FUNCTION_BLOCK Q_GraphicsContext (* Command Graphics Context ( Part 6 - F.56 ) *)
  (* Standard: ISO 11783-6; Description: Copyright (c) 2022 HR Agrartechnik GmbH This program and the accompanying materials are made available under the terms of the Eclipse Public License 2.0 which is available at https://www.eclipse.org/legal/epl-2.0/ SPDX-License-Identifier: EPL-2.0 see Description Tab *)
  (* Version 1.0, 2022-07-08, Franz Höpfinger, HR Agrartechnik GmbH *)
  PACKAGE isobus::UT::Q;
  IMPORT eclipse4diac::core::TypeHash;
  IMPORT isobus::UT::Q::IDs::ID_NULL;
  (* Documentation:
  Command Graphics Context ( Part 6 - F.56 )
   This command is used to manipulate a graphics Context object (only on version 4 or later VTs).
   param[in] {objectID, uint16_t}
   Object ID of a Graphics Context object
   param[in] {SubCommandID, uint8_t}
   Sub-Command ID
   param[in] {ParameterSubCommandID_Byte, const uint8_t *}
   Parameters based on sub-command ID byte
   param[in] {LenBytes, uint16_t}
   Length in bytes of parameter list
   Return Values: 
   int16_t
    - VT_E_NO_ERR (0) - OK
   - VT_E_OVERFLOW (-6) - buffer overflow
   - VT_E_NOACT (-8) - Command not possible in current state
   - VT_E_NO_INSTANCE (-21) - No VT client available
   - VT_E_ISO_INSTANCE_INVALID (-129) - Identifier for instance (connection) invalid
   - VT_E_NOT_ALIVE (-130) - Identifier for instance valid, but VT Dead.
    Note
    - Function uses string buffer ( Parameterlist has to be smaller than ISO_VTC_CMD_STR_MAX_LENGTH )
  *)
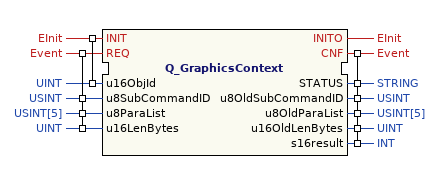
  EVENT_INPUT
    INIT : EInit WITH u16ObjId; (* Service Initialization *)
    REQ WITH u8SubCommandID, u8ParaList, u16LenBytes; (* Service Request *)
  END_EVENT
  EVENT_OUTPUT
    INITO : EInit; (* Initialization Confirm *)
    CNF WITH STATUS, s16result, u8OldSubCommandID, u8OldParaList, u16OldLenBytes; (* Confirmation of Requested Service *)
  END_EVENT
  VAR_INPUT
    u16ObjId : UINT := ID_NULL; (* Object ID *)
    u8SubCommandID : USINT; (* Sub-Command ID *)
    u8ParaList : ARRAY [0..4] OF USINT; (* Parameters based on sub-command ID byte *)
    u16LenBytes : UINT; (* Length in bytes of parameter list *)
  END_VAR
  VAR_OUTPUT
    STATUS : STRING; (* Service Status *)
    u8OldSubCommandID : USINT; (* Old Sub-Command ID *)
    u8OldParaList : ARRAY [0..4] OF USINT; (* Old parameters based on sub-command ID byte *)
    u16OldLenBytes : UINT; (* Old length in bytes of parameter list *)
    s16result : INT; (* retval see description *)
  END_VAR
END_FUNCTION_BLOCK
